(* Logix 5000 project; controller KTC_LAB7_PART2 vendor 1 type 14 code 150 rev 30.11; software revision 30.00 *)

TASK MainTask (continuous, watchdog 500 ms) : MainProgram

MODULES
   Local : vendor 1 type 14 code 150 (Compact 0, rev 30.11)
      Counters : Embedded (Compact 3, rev 1.1, Output RPI 20 ms)
      Discrete_IO : Embedded (Compact 1, rev 3.1, Output RPI 20 ms)
      Analog_IO : Embedded (Compact 2, rev 1.1, Output RPI 80 ms)
END_MODULES

PROGRAM MainProgram   (* main routine MainRoutine *)
VAR
   pl0 : ALIAS FOR Local:1:O.Data.11;   // red
   pl1 : ALIAS FOR Local:1:O.Data.3;   // green
   pl2 : ALIAS FOR Local:1:O.Data.7;   // yellow
   T4_0 : TIMER := (PRE := 15000, ACC := 13477, EN := 1, TT := 1);
   T4_1 : TIMER := (PRE := 10000);
   T4_2 : TIMER := (PRE := 5000);
END_VAR

ROUTINE MainRoutine   (* ladder *)
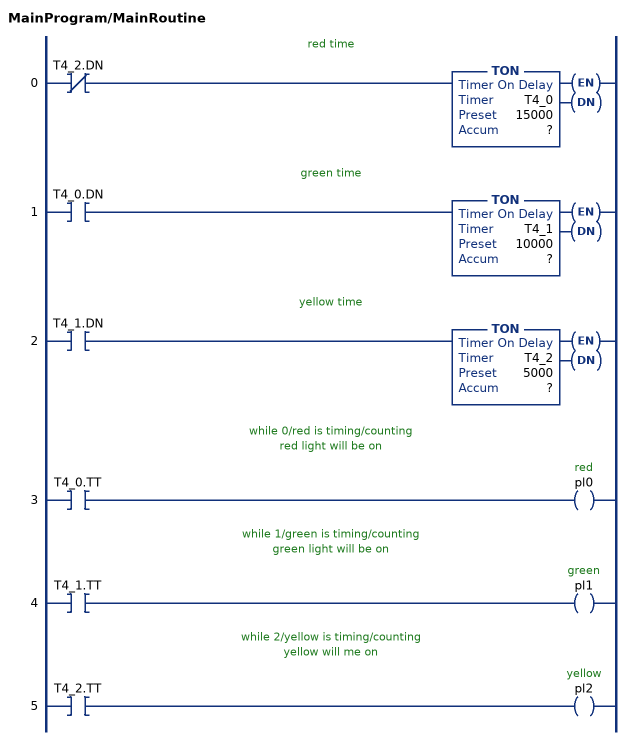
   // red time
   0: XIO(T4_2.DN)TON(T4_0,?,?);
   // green time
   1: XIC(T4_0.DN)TON(T4_1,?,?);
   // yellow time
   2: XIC(T4_1.DN)TON(T4_2,?,?);
   // while 0/red is timing/counting
   // red light will be on
   3: XIC(T4_0.TT)OTE(pl0);
   // while 1/green is timing/counting
   // green light will be on
   4: XIC(T4_1.TT)OTE(pl1);
   // while 2/yellow is timing/counting
   // yellow will me on
   5: XIC(T4_2.TT)OTE(pl2);
END_ROUTINE
END_PROGRAM
